Staubli VAL3: trajBuffer.pgx

public program trajBuffer(num x_nElems, num x_nPtsPopped)
begin

  // update trajectory buffer size

  gotoxy(scMonitor, 0,3)
  // 18 characteres: gotoxy(19,3) to insert status
  put(scMonitor, "Trajectory buffer:")
  gotoxy(scMonitor, 19,3)
  put(scMonitor, x_nElems)
  // also print number of points popped from buffer
  gotoxy(scMonitor, 24,3)
  put(scMonitor, x_nPtsPopped)

end
